{attribute 'linkalways'} 
{attribute 'no_explicit_call' := 'This FB is a CLASS and must be accessed using methods or properties'}
{attribute 'enable_dynamic_creation'}
FUNCTION_BLOCK _WORD EXTENDS NumericDatatypeBase IMPLEMENTS I_WORD
VAR
	localData : WORD;
	activeData : REFERENCE TO WORD REF= localData;
END_VAR

PROPERTY PUBLIC Address : PVOID
GET
Address := ADR(activeData);
END_GET
END_PROPERTY

METHOD PUBLIC ClearReference
VAR_INPUT
END_VAR
activeData REF= localData;
END_METHOD

METHOD PUBLIC Clone : I_Datatype
VAR
    pClone : POINTER TO _WORD;
END_VAR
pClone := __NEW(_WORD(InitialValue := Value));
Clone := pClone^;
END_METHOD

METHOD FB_init : BOOL
VAR_INPUT
	bInitRetains : BOOL; // if TRUE, the retain variables are initialized (warm start / cold start)
	bInCopyCode : BOOL;  // if TRUE, the instance afterwards gets moved WORDo the copy code (online change)
	InitialValue : WORD;
END_VAR
localData := InitialValue;
END_METHOD

PROPERTY PUBLIC IsEven : BOOL
GET
IsEven := (Value mod 2) = 0;
END_GET
END_PROPERTY

PROPERTY PUBLIC IsFloat : BOOL
GET
IsFloat := FALSE;
END_GET
END_PROPERTY

PROPERTY PUBLIC IsSigned : BOOL
GET
IsSigned := FALSE;
END_GET
END_PROPERTY

METHOD PUBLIC MakeReferenceTo
VAR_INPUT
	ReferenceTarget : REFERENCE TO WORD;
END_VAR
activeData REF= ReferenceTarget;
END_METHOD

PROPERTY PUBLIC MaxValue : WORD
GET
MaxValue :=  DatatypeLimits.WORD_MAX_VALUE;
END_GET
END_PROPERTY

PROPERTY PUBLIC MinValue : WORD
GET
MinValue := DatatypeLimits.WORD_MIN_VALUE;
END_GET
END_PROPERTY

METHOD PROTECTED SerializeMaxValue
VAR_INPUT
	Serializer : I_Serializer;
END_VAR
Serializer.AddWord(MaxValue);
END_METHOD

METHOD PROTECTED SerializeMinValue
VAR_INPUT
	Serializer : I_Serializer;
END_VAR
Serializer.AddWord(MinValue);
END_METHOD

METHOD PUBLIC SerializeWith
VAR_INPUT
	Serializer : I_Serializer;
END_VAR
Serializer.AddWord(activeData);
END_METHOD

PROPERTY PUBLIC Size : UDINT
GET
Size := SIZEOF(activeData);
END_GET
END_PROPERTY

METHOD PUBLIC TryConvertTo : BOOL
VAR_INPUT
	Destination : ANY;
END_VAR
TryConvertTo := TryConvert_WORD_TO_Destination(activeData, Destination);
END_METHOD

METHOD PUBLIC TryConvertTo_ : BOOL
VAR_INPUT
	Destination : I_Datatype;
END_VAR
VAR
	resultofBitConversion : BOOL;
	destinationAs_BIT : I_BIT;
	destinationAs_BOOL : I_BOOL;
	destinationAs_BYTE : I_BYTE;
	destinationAs_DINT : I_DINT;
	destinationAs_DT : I_DT;
	destinationAs_DWORD : I_DWORD;
	destinationAs_INT : I_INT;
	destinationAs_LINT : I_LINT;
	destinationAs_LREAL : I_LREAL;
	destinationAs_LWORD : I_LWORD;
	destinationAs_REAL : I_REAL;
	destinationAs_SINT : I_SINT;
	destinationAs_STRING : I_STRING;
	destinationAs_TOD : I_TOD;
	destinationAs_UDINT : I_UDINT;
	destinationAs_UINT : I_UINT;
	destinationAs_ULINT : I_ULINT;
	destinationAs_USINT : I_USINT;
	destinationAs_WORD : I_WORD;
END_VAR
IF destination.TryResolveAs_BIT(destinationAs_BIT) AND_THEN TryConvert_WORD_TO_BOOL(activeData, resultofBitConversion) THEN
	destinationAs_BIT.Value := resultOfBitConversion;
	TryConvertTo_ := TRUE;
	RETURN;
END_IF

IF destination.TryResolveAs_BOOL(destinationAs_BOOL) THEN
	TryConvertTo_ := TryConvert_WORD_TO_BOOL(activeData, destinationAs_BOOL.Value);
	RETURN;
END_IF
		
IF destination.TryResolveAs_BYTE(destinationAs_BYTE) THEN
	TryConvertTo_ := TryConvert_WORD_TO_BYTE(activeData, destinationAs_BYTE.Value);
	RETURN;
END_IF

IF destination.TryResolveAs_DINT(destinationAs_DINT) THEN
	TryConvertTo_ := TryConvert_WORD_TO_DINT(activeData, destinationAs_DINT.Value);
	RETURN;
END_IF

IF destination.TryResolveAs_DT(destinationAs_DT) THEN
	TryConvertTo_ := TryConvert_WORD_TO_DT(activeData, destinationAs_DT.Value);
	RETURN;
END_IF

IF destination.TryResolveAs_DWORD(destinationAs_DWORD) THEN
	TryConvertTo_ := TryConvert_WORD_TO_DWORD(activeData, destinationAs_DWORD.Value);
	RETURN;
END_IF

IF destination.TryResolveAs_INT(destinationAs_INT) THEN
	TryConvertTo_ := TryConvert_WORD_TO_INT(activeData, destinationAs_INT.Value);
	RETURN;
END_IF

IF destination.TryResolveAs_LINT(destinationAs_LINT) THEN
	TryConvertTo_ := TryConvert_WORD_TO_LINT(activeData, destinationAs_LINT.Value);
	RETURN;
END_IF

IF destination.TryResolveAs_LREAL(destinationAs_LREAL) THEN
	TryConvertTo_ := TryConvert_WORD_TO_LREAL(activeData, destinationAs_LREAL.Value);
	RETURN;
END_IF

IF destination.TryResolveAs_LWORD(destinationAs_LWORD) THEN
	TryConvertTo_ := TryConvert_WORD_TO_LWORD(activeData, destinationAs_LWORD.Value);
	RETURN;
END_IF

IF destination.TryResolveAs_REAL(destinationAs_REAL) THEN
	TryConvertTo_ := TryConvert_WORD_TO_REAL(activeData, destinationAs_REAL.Value);
	RETURN;
END_IF

IF destination.TryResolveAs_SINT(destinationAs_SINT) THEN
	TryConvertTo_ := TryConvert_WORD_TO_SINT(activeData, destinationAs_SINT.Value);
	RETURN;
END_IF

IF destination.TryResolveAs_STRING(destinationAs_STRING) THEN
	TryConvertTo_ := TryConvert_WORD_TO_STRING(activeData, destinationAs_STRING.Value);
	RETURN;
END_IF

IF destination.TryResolveAs_TOD(destinationAs_TOD) THEN
	TryConvertTo_ := TryConvert_WORD_TO_TOD(activeData, destinationAs_TOD.Value);
	RETURN;
END_IF

IF destination.TryResolveAs_UDINT(destinationAs_UDINT) THEN
	TryConvertTo_ := TryConvert_WORD_TO_UDINT(activeData, destinationAs_UDINT.Value);
	RETURN;
END_IF

IF destination.TryResolveAs_UINT(destinationAs_UINT) THEN
	TryConvertTo_ := TryConvert_WORD_TO_UINT(activeData, destinationAs_UINT.Value);
	RETURN;
END_IF

IF destination.TryResolveAs_ULINT(destinationAs_ULINT) THEN
	TryConvertTo_ := TryConvert_WORD_TO_ULINT(activeData, destinationAs_ULINT.Value);
	RETURN;
END_IF

IF destination.TryResolveAs_USINT(destinationAs_USINT) THEN
	TryConvertTo_ := TryConvert_WORD_TO_USINT(activeData, destinationAs_USINT.Value);
	RETURN;
END_IF

IF destination.TryResolveAs_WORD(destinationAs_WORD) THEN
	TryConvertTo_ := TryConvert_WORD_TO_WORD(activeData, destinationAs_WORD.Value);
	RETURN;
END_IF
END_METHOD

METHOD TryDeserializeFrom : BOOL
VAR_INPUT
	Deserializer : I_Deserializer;
	Feedback : I_DeserializerFeedback;
END_VAR
TryDeserializeFrom := Deserializer.TryGetWord(activeData, Feedback);
END_METHOD

METHOD TryMakeReferenceTo : BOOL
VAR_INPUT
	Target : I_Datatype;
END_VAR
VAR
	pTargetData : POINTER TO WORD;
END_VAR
IF NOT IsEquivalentTo(Target) THEN
	RETURN;
END_IF

pTargetData := Target.Address;
activeData REF= pTargetData^;
TryMakeReferenceTo := TRUE;
END_METHOD

METHOD PUBLIC TryResolveAs_WORD : BOOL
VAR_INPUT
	Destination : REFERENCE TO I_WORD;
END_VAR
Destination := THIS^;
TryResolveAs_WORD := TRUE;
END_METHOD

PROPERTY PUBLIC TypeName : T_MAXSTRING
GET
TypeName := 'WORD';
END_GET
END_PROPERTY

{warning disable C5410}
PROPERTY PUBLIC Value : REFERENCE TO WORD
{warning restore C5410}
GET
Value REF= activeData;
END_GET
END_PROPERTY

END_FUNCTION_BLOCK

(* stored: Version 1.1.0.1, ProductVersion 3.1.4024.15
   POU _WORD: Id {785b4543-75b4-4d22-ba61-129866dbb78f}, SpecialFunc None
   Folder Constructor: Id {2bc942c9-15ef-443c-86a0-0ba3d6f8acbf}
   Folder Protected: Id {a63c5a23-6486-48b9-8570-ceb36a757b18}
   Property Address: Id {dde93b64-d15e-4c83-a1c7-9a71a5203dbd}
   Get Get: Id {15831d15-e22a-4e2b-bf87-eb7a5f0007f2}
   Method ClearReference: Id {006bc84c-7a71-4a67-9fcd-5c4ef11d0d04}
   Method Clone: Id {3ad80d2a-a76e-4b25-a839-a3445f1727ce}
   Method FB_init: Id {25cb8094-357a-4e3b-b5fe-15624aba575c}
   Property IsEven: Id {9e740dfe-6f0d-0e02-2109-625bfe544a0f}
   Get Get: Id {9d1a7e75-20cb-0222-3716-8a44a1b6f195}
   Property IsFloat: Id {9031cfa6-6438-4d3a-94a7-7b1d37055da1}
   Get Get: Id {7390886d-ad43-4baa-ba6b-c5b294a25c3a}
   Property IsSigned: Id {75ebcade-d7b4-4897-8091-d07bca5214dc}
   Get Get: Id {4bd4aebb-55aa-4478-8ca6-2f0f9370ffc2}
   Method MakeReferenceTo: Id {4c888c95-4902-445b-bffe-15128e43a6d3}
   Property MaxValue: Id {df183709-e5a2-44ff-87d7-9368105dab63}
   Get Get: Id {28fd4b6d-ce35-4c59-a813-06cb5556e621}
   Property MinValue: Id {37d80b64-8e58-4f9d-9f8a-37a1acd57600}
   Get Get: Id {788b7e61-0ffc-4237-a55d-41150ae7f999}
   Method SerializeMaxValue: Id {6cf67daa-fa5f-4f6b-b5c0-6a8a33d5e532}
   Method SerializeMinValue: Id {9e6ebab6-c168-44a3-9857-d853802e8cef}
   Method SerializeWith: Id {ff03b8e8-977c-4201-aaa1-7b0e153d93cd}
   Property Size: Id {2bdd1b22-de81-4397-8b38-532f4fd909a3}
   Get Get: Id {b95c9a04-8956-463c-ac0e-bd89d4a7164f}
   Method TryConvertTo: Id {21b44d84-eba9-0892-1d7e-06dadc3ac35b}
   Method TryConvertTo_: Id {13255a93-2560-047a-0453-50e24cb15db1}
   Method TryDeserializeFrom: Id {00f03103-9e65-4c26-99af-92a5fda659ca}
   Method TryMakeReferenceTo: Id {a85aab6e-0868-49b5-a56c-8d1f3422f73f}
   Method TryResolveAs_WORD: Id {a8056bec-2148-06c1-1b1e-7efe596855ba}
   Property TypeName: Id {ea67172d-3b40-4ad0-ae37-3ab08a0b7855}
   Get Get: Id {b997ca83-025a-40c6-96c4-34086c410ab4}
   Property Value: Id {e62bcf86-3880-4080-9eae-bbad242889c9}
   Get Get: Id {466faa1b-1333-47fa-aaf0-4b401c13734f} *)
